{attribute 'qualified_only'}
VAR_GLOBAL
	nGANTRY_TOLERANCE_NM_DEFAULT : LINT := 50000; // default gantry tolerance in encoder counts = nm
END_VAR

(* stored: Version 1.1.0.1, ProductVersion 3.1.4022.12
   GVL GVL_HOMS: Id {7aa67172-25b3-4e6c-90f4-628372b0226d} *)
